// TIA Portal project "PID_TANK1_TANK2" (V16)

(* hardware
DEVICE "S7-1200 station_1"  S7-1200 Station
   slot 0: "Rack_0"  S7-1200 Rack  Rack  V1.0
   slot 1: "PLC_1"  CPU 1214C DC/DC/DC  6ES7 214-1AG40-0XB0  V4.2
   slot 2: "AI 4x13BIT/AQ 2x14BIT_1"  6ES7 234-4HE32-0XB0  V2.1
*)

// ===== PLC "PLC_1"  CPU 1214C DC/DC/DC =====

VAR_GLOBAL   // PLC tag table "Default tag table"
   "StartPump1" AT %I0.0 : Bool;
   "Stop1" AT %I0.1 : Bool;
   "Pump1 M" AT %Q0.0 : Bool;
   "Level Tank 1" AT %IW64 : Int;
   "Level Tank1 Memory" AT %MD2 : Real;
   "Level Tank 2" AT %IW66 : Int;
   "Level Tank2 Memory" AT %MD4 : Real;
   "MV DATA T1 01" AT %MD6 : Real;
   "MV DATA T1 02" AT %MD8 : Real;
   "PUMP1" AT %QW98 : Int;
   "Tag_1" AT %QW96 : Int;
   "Setpoint Tank2" AT %MW10 : Int;
END_VAR

DATA_BLOCK "Data_PID"   // DB3
{ S7_Optimized_Access := 'FALSE' }
VERSION : 0.1
   VAR
      "SP TANK2" : Real := 0.0;
      "PV TANK1" : Real;
      "PV TANK2" : Real;
      "MV TANK1" : Real;
      "MV TANK2" : Real;
      "PV TANK1 d" : Word;
      "PV TANK2 d" : Word;
      "SP TANK2 d" : Word;
   END_VAR
BEGIN
END_DATA_BLOCK

FUNCTION "Scale" : Void   // FC2, LAD
{ S7_Optimized_Access := 'TRUE' }
VERSION : 0.1
BEGIN

REGION Network 1: SETPOINT
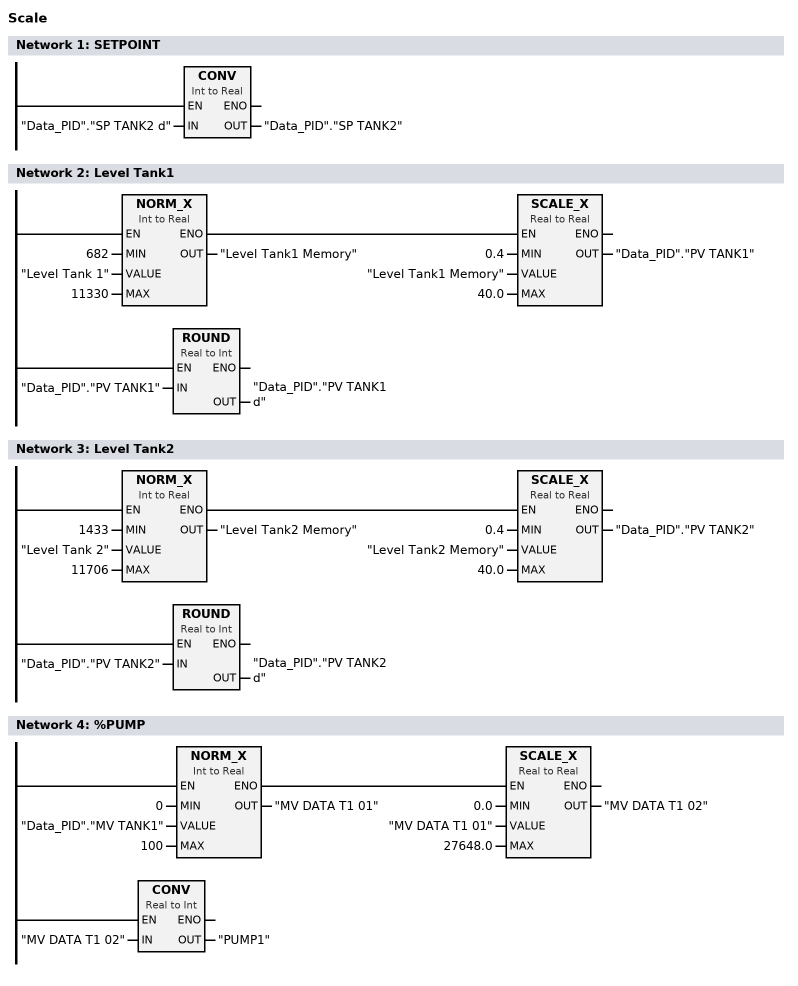
   RUNG wire#powerrail
      { S7_Templates := "[SrcType := Int, DestType := Real]" } Convert(in := "Data_PID"."SP TANK2 d", out => "Data_PID"."SP TANK2")
   END_RUNG
   // the same network as SCL:
   "Data_PID"."SP TANK2" := INT_TO_REAL("Data_PID"."SP TANK2 d");
END_REGION

REGION Network 2: Level Tank1
   RUNG wire#powerrail
      { S7_Templates := "[SrcType := Int, DestType := Real]" } Normalize(min := 682, value := "Level Tank 1", max := 11330, out => "Level Tank1 Memory")
      { S7_Templates := "[SrcType := Real, DestType := Real]" } Scale(min := 0.4, value := "Level Tank1 Memory", max := 40.0, out => "Data_PID"."PV TANK1")
   END_RUNG
   RUNG wire#powerrail
      { S7_Templates := "[SrcType := Real, DestType := Int]" } Round(in := "Data_PID"."PV TANK1", out => "Data_PID"."PV TANK1 d")
   END_RUNG
   // the same network as SCL:
   "Level Tank1 Memory" := NORM_X(MIN := 682, VALUE := "Level Tank 1", MAX := 11330);
   "Data_PID"."PV TANK1" := SCALE_X(MIN := 0.4, VALUE := "Level Tank1 Memory", MAX := 40.0);
   "Data_PID"."PV TANK1 d" := ROUND("Data_PID"."PV TANK1");
END_REGION

REGION Network 3: Level Tank2
   RUNG wire#powerrail
      { S7_Templates := "[SrcType := Int, DestType := Real]" } Normalize(min := 1433, value := "Level Tank 2", max := 11706, out => "Level Tank2 Memory")
      { S7_Templates := "[SrcType := Real, DestType := Real]" } Scale(min := 0.4, value := "Level Tank2 Memory", max := 40.0, out => "Data_PID"."PV TANK2")
   END_RUNG
   RUNG wire#powerrail
      { S7_Templates := "[SrcType := Real, DestType := Int]" } Round(in := "Data_PID"."PV TANK2", out => "Data_PID"."PV TANK2 d")
   END_RUNG
   // the same network as SCL:
   "Level Tank2 Memory" := NORM_X(MIN := 1433, VALUE := "Level Tank 2", MAX := 11706);
   "Data_PID"."PV TANK2" := SCALE_X(MIN := 0.4, VALUE := "Level Tank2 Memory", MAX := 40.0);
   "Data_PID"."PV TANK2 d" := ROUND("Data_PID"."PV TANK2");
END_REGION

REGION Network 4: %PUMP
   RUNG wire#powerrail
      { S7_Templates := "[SrcType := Int, DestType := Real]" } Normalize(min := 0, value := "Data_PID"."MV TANK1", max := 100, out => "MV DATA T1 01")
      { S7_Templates := "[SrcType := Real, DestType := Real]" } Scale(min := 0.0, value := "MV DATA T1 01", max := 27648.0, out => "MV DATA T1 02")
   END_RUNG
   RUNG wire#powerrail
      { S7_Templates := "[SrcType := Real, DestType := Int]" } Convert(in := "MV DATA T1 02", out => "PUMP1")
   END_RUNG
   // the same network as SCL:
   "MV DATA T1 01" := NORM_X(MIN := 0, VALUE := "Data_PID"."MV TANK1", MAX := 100);
   "MV DATA T1 02" := SCALE_X(MIN := 0.0, VALUE := "MV DATA T1 01", MAX := 27648.0);
   "PUMP1" := REAL_TO_INT("MV DATA T1 02");
END_REGION
END_FUNCTION

ORGANIZATION_BLOCK "Main"   // OB1, LAD, ProgramCycle
TITLE = "Main Program Sweep (Cycle)"
{ S7_Optimized_Access := 'TRUE' }
VERSION : 0.1
   VAR_INPUT
      Initial_Call : Bool;   // Initial call of this OB
      Remanence : Bool;   // =True, if remanent data are available
   END_VAR
BEGIN

REGION Network 1
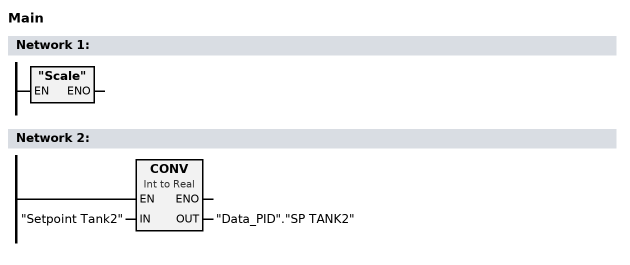
   RUNG wire#powerrail
      "Scale"()
   END_RUNG
   // the same network as SCL:
   "Scale"();
END_REGION

REGION Network 2
   RUNG wire#powerrail
      { S7_Templates := "[SrcType := Int, DestType := Real]" } Convert(in := "Setpoint Tank2", out => "Data_PID"."SP TANK2")
   END_RUNG
   // the same network as SCL:
   "Data_PID"."SP TANK2" := INT_TO_REAL("Setpoint Tank2");
END_REGION
END_ORGANIZATION_BLOCK

ORGANIZATION_BLOCK "Cyclic interrupt"   // OB30, LAD, CyclicInterrupt
{ S7_Optimized_Access := 'TRUE' }
VERSION : 0.1
   VAR_INPUT
      Initial_Call : Bool;   // Initial call of this OB
      Event_Count : Int;   // Events discarded
   END_VAR
BEGIN

REGION Network 1
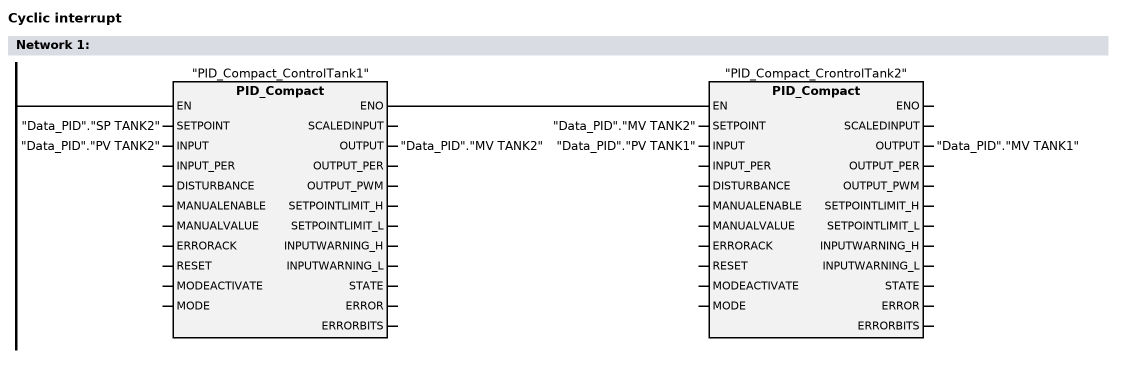
   // ENO of a box is taken as its EN; it also drops when the box reports an error
   "PID_Compact_ControlTank1"(Setpoint := "Data_PID"."SP TANK2",   // PID_Compact
                           Input := "Data_PID"."PV TANK2",
                           Output => "Data_PID"."MV TANK2");
   "PID_Compact_CrontrolTank2"(Setpoint := "Data_PID"."MV TANK2",   // PID_Compact
                           Input := "Data_PID"."PV TANK1",
                           Output => "Data_PID"."MV TANK1");
END_REGION
END_ORGANIZATION_BLOCK